FUNCTION_BLOCK FB_Washing
VAR_INPUT
	bExecute		: BOOL;
END_VAR
VAR_OUTPUT
	bDone			: BOOL;
	bError			: BOOL;
	wErrorID		: BOOL;
END_VAR
VAR
	
END_VAR

END_FUNCTION_BLOCK

(* stored: Version 1.1.0.1, ProductVersion 3.1.4024.11
   POU FB_Washing: Id {c44c8330-ba9b-44dc-b7d6-2c009118cac6}, SpecialFunc None *)
